FUNCTION_BLOCK CfbTlNetwork
  (* Standard: 61499-2 *)
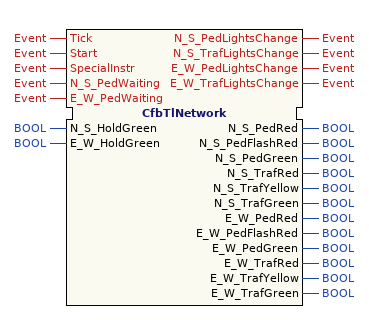
  EVENT_INPUT
    Tick;
    Start;
    SpecialInstr;
    N_S_PedWaiting;
    E_W_PedWaiting;
  END_EVENT
  EVENT_OUTPUT
    N_S_PedLightsChange;
    N_S_TrafLightsChange;
    E_W_PedLightsChange;
    E_W_TrafLightsChange;
  END_EVENT
  VAR_INPUT
    N_S_HoldGreen : BOOL;
    E_W_HoldGreen : BOOL;
  END_VAR
  VAR_OUTPUT
    N_S_PedRed : BOOL;
    N_S_PedFlashRed : BOOL;
    N_S_PedGreen : BOOL;
    N_S_TrafRed : BOOL;
    N_S_TrafYellow : BOOL;
    N_S_TrafGreen : BOOL;
    E_W_PedRed : BOOL;
    E_W_PedFlashRed : BOOL;
    E_W_PedGreen : BOOL;
    E_W_TrafRed : BOOL;
    E_W_TrafYellow : BOOL;
    E_W_TrafGreen : BOOL;
  END_VAR
  FBS
    N_S : CfbOneLink;
    E_W : CfbOneLink;
    mt : BfbIntersectionMutex;
  END_FBS
  EVENT_CONNECTIONS
    Tick TO N_S.Tick;
    Tick TO E_W.Tick;
    SpecialInstr TO N_S.SpecialInstr;
    SpecialInstr TO E_W.SpecialInstr;
    Start TO mt.Start;
    mt.N_S_Start TO N_S.GoSeq;
    N_S.DoneSeq TO mt.N_S_Done;
    mt.E_W_Start TO E_W.GoSeq;
    E_W.DoneSeq TO mt.E_W_Done;
    N_S_PedWaiting TO N_S.PedWaiting;
    E_W_PedWaiting TO E_W.PedWaiting;
    N_S.PedLightsChange TO N_S_PedLightsChange;
    N_S.TrafLightsChange TO N_S_TrafLightsChange;
    E_W.PedLightsChange TO E_W_PedLightsChange;
    E_W.TrafLightsChange TO E_W_TrafLightsChange;
  END_CONNECTIONS
  DATA_CONNECTIONS
    N_S_HoldGreen TO N_S.HoldGreen;
    E_W_HoldGreen TO E_W.HoldGreen;
    N_S.PedRed TO N_S_PedRed;
    N_S.PedFlashRed TO N_S_PedFlashRed;
    N_S.PedGreen TO N_S_PedGreen;
    N_S.TrafRed TO N_S_TrafRed;
    N_S.TrafYellow TO N_S_TrafYellow;
    N_S.TrafGreen TO N_S_TrafGreen;
    E_W.PedRed TO E_W_PedRed;
    E_W.PedFlashRed TO E_W_PedFlashRed;
    E_W.PedGreen TO E_W_PedGreen;
    E_W.TrafRed TO E_W_TrafRed;
    E_W.TrafYellow TO E_W_TrafYellow;
    E_W.TrafGreen TO E_W_TrafGreen;
  END_CONNECTIONS
END_FUNCTION_BLOCK
